FUNCTION_BLOCK FB_Stromzaehler_BHKW
VAR_INPUT
	Telegramm	: ARRAY[1..cMBUS_MaxTelegrams] OF ST_MBus_Data2;

END_VAR
VAR_IN_OUT
	Zustand		: ST_SZ_Zustand;
END_VAR
VAR
END_VAR
VAR // added by the converter: edge detectors and wires of the graphical bodies
    _w1, _w2 : ANY;
END_VAR

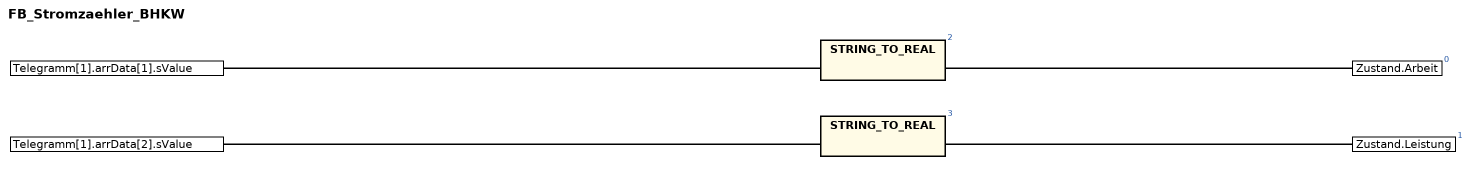
Zustand.Arbeit := _w1;
Zustand.Leistung := _w2;
_w1 := STRING_TO_REAL(Telegramm[1].arrData[1].sValue);
_w2 := STRING_TO_REAL(Telegramm[1].arrData[2].sValue);

END_FUNCTION_BLOCK

(* stored: Version 1.1.0.1, ProductVersion 3.1.4024.9
   POU FB_Stromzaehler_BHKW: Id {bf48f9d0-7fa0-4792-ac10-22b6142522f5}, SpecialFunc None *)
